// TwinCAT 3 PLC project TcUnit_Tests
// ProgramVersion: 3.1.4024.12
// libraries:
//   Tc2_Standard, * (Beckhoff Automation GmbH)
//   Tc2_System, * (Beckhoff Automation GmbH)
//   Tc3_Module, * (Beckhoff Automation GmbH)
//   TcUnit, * (www.tcunit.org)
// project tree:
//   / PlcTask.TcTTO
//   Tests/ FB_FanControl_Test.TcPOU, FC_HeatingCurve_Test.TcPOU, PRG_TEST.TcPOU

CONFIGURATION TcUnit_Tests
    RESOURCE PLC ON TwinCAT3
        TASK PlcTask(INTERVAL := T#10ms, PRIORITY := 20);
        PROGRAM PRG_TEST WITH PlcTask : PRG_TEST;
    END_RESOURCE
END_CONFIGURATION

// ---- Tests/PRG_TEST.TcPOU
PROGRAM PRG_TEST
VAR
	HeatingCurve_Test : FC_HeatingCurve_Test;
	FanControlTest : FB_FanControl_Test;
END_VAR

TcUnit.RUN();

END_PROGRAM

// ---- Tests/FC_HeatingCurve_Test.TcPOU
FUNCTION_BLOCK FC_HeatingCurve_Test EXTENDS FB_TestSuite
VAR

END_VAR

TAmbNegative();
TAmbZero();
HeatingCurveZero();
HeatingCurveNegative();

METHOD HeatingCurveNegative // This method checks whether the heating curve can have a negative value
VAR
	HeatingCurveRes: Real;		//Actual value for Heating Curve
	ExpectedValue : REAL := -1;	//Expected value for Heating Curve
	fSlope: REAL := -1;				//Slope of Heating Curve
	fOffset: REAL := 35;				//Offset of Heating Curve

END_VAR
TEST('HeatingCurveNegative');
 
HeatingCurveRes := FC_HeatingCurve(fTempAmb := 36, fSlope, fOffset);
 
AssertEquals(Expected := ExpectedValue,
             Actual := HeatingCurveRes,
             Message := 'The calculation is not correct');
 
TEST_FINISHED();
END_METHOD

METHOD HeatingCurveZero // This method checks whether the heating curve can have zero as value
VAR
	HeatingCurveRes: REAL;		//Actual value for Heating Curve
	ExpectedValue : REAL := 0;  //Expected value for Heating Curve
	fSlope: REAL := -1;				//Slope of Heating Curve
	fOffset: REAL := 35;				//Offset of Heating Curve
//	fTempAmb: REAL

END_VAR
TEST('HeatingCurveZero');
 
HeatingCurveRes := FC_HeatingCurve(fTempAmb := 35, fSlope, fOffset);
 
AssertEquals(Expected := ExpectedValue,
             Actual := HeatingCurveRes,
             Message := 'The calculation is not correct');
 
TEST_FINISHED();
END_METHOD

METHOD TAmbNegative // This method checks whether negative ambient temperatures work properly
VAR
	HeatingCurveRes: REAL;		 //Actual value for Heating Curve
	ExpectedValue : REAL := 40;  //Expected value for Heating Curve
	fSlope: REAL := -1;				 //Slope of Heating Curve
	fOffset: REAL := 35;				 //Offset of Heating Curve
END_VAR
TEST('TAmbNegative');
 
HeatingCurveRes := FC_HeatingCurve(fTempAmb := -5, fSlope, fOffset);
 
AssertEquals(Expected := ExpectedValue,
             Actual := HeatingCurveRes,
             Message := 'The calculation is not correct');
 
TEST_FINISHED();
END_METHOD

METHOD TAmbZero // This method checks whether zero degrees as ambient temperature work properly
VAR
	HeatingCurveRes : REAL;		  //Actual value for Heating Curve
	ExpectedValue : REAL := 35;   //Expected value for Heating Curve
	fSlope: REAL := -1;				  //Slope of Heating Curve	
	fOffset: REAL := 35;				  //Offset of Heating Curve

END_VAR
TEST('TAmbZero');
 
HeatingCurveRes := FC_HeatingCurve(fTempAmb := 0, fSlope, fOffset);
 
AssertEquals(Expected := ExpectedValue,
             Actual := HeatingCurveRes,
             Message := 'The calculation is not correct');
 
TEST_FINISHED();
END_METHOD

END_FUNCTION_BLOCK

// ---- Tests/FB_FanControl_Test.TcPOU
FUNCTION_BLOCK FB_FanControl_Test EXTENDS FB_TestSuite
VAR
END_VAR

METHOD FanSpeedMax
VAR
	FanControlRes: REAL;			//Actual value of FanControl
	ExpectedValue : REAL := 100;	//Expected value for FanControl

END_VAR
TEST('FanSpeedZero');
 
FanControlRes := FB_FanControl(fSpeed := 327.67);
 
AssertEquals(Expected := ExpectedValue,
             Actual := FanControlRes,
             Message := 'The calculation is not correct');
 
TEST_FINISHED();
END_METHOD

METHOD FanSpeedZero
VAR
	FanControlRes: REAL;		//Actual value of FanControl
	ExpectedValue : REAL := 0;	//Expected value for FanControl

END_VAR
TEST('FanSpeedZero');
 
FanControlRes := FB_FanControl(fSpeed := 0);
 
AssertEquals(Expected := ExpectedValue,
             Actual := FanControlRes,
             Message := 'The calculation is not correct');
 
TEST_FINISHED();
END_METHOD

END_FUNCTION_BLOCK
